{attribute 'GeneratedUsingTerminal: KL8610-0004'}
{attribute addProperty BoxType "KL8610-0004"}
{attribute addProperty Id "KL8601_1AT %Q*KL_6576A6810KL8601_2AT %Q*KL_6576A6810KL8601_3AT %Q*KL_6576A6810KL8601_4AT %Q*KL_6576A6810KL8601_5AT %Q*KL_6576A6810"}
{attribute addProperty CRC "925658092"}
{attribute addProperty Size "0"}
TYPE KL_372C6BEC :
STRUCT
	{attribute addProperty Name "KL8601_1"}
	KL8601_1 : KL_6576A681;
	{attribute addProperty Name "KL8601_2"}
	KL8601_2 : KL_6576A681;
	{attribute addProperty Name "KL8601_3"}
	KL8601_3 : KL_6576A681;
	{attribute addProperty Name "KL8601_4"}
	KL8601_4 : KL_6576A681;
	{attribute addProperty Name "KL8601_5"}
	KL8601_5 : KL_6576A681;
END_STRUCT
END_TYPE

(* stored: Version 1.2.0.0, ProductVersion 3.1.4024.9
   DUT KL_372C6BEC: Id {8d3cb635-4f9c-4a61-8106-d5a48ad92911} *)
